Omron CX-Programmer project NewProject (CX-Programmer 9.73)

# PLC NewPLC1: CP1E N20

## Global symbols (name address type ; comment)
0.01 BOOL  ; PB START
100.00 BOOL  ; OUTPUT
100.04 BOOL  ; OUTPUT 2
T001 BOOL  ; TIMER
T002 BOOL  ; TIMER2

## Program NewProgram1 (cyclic task 0)

### Section Section1

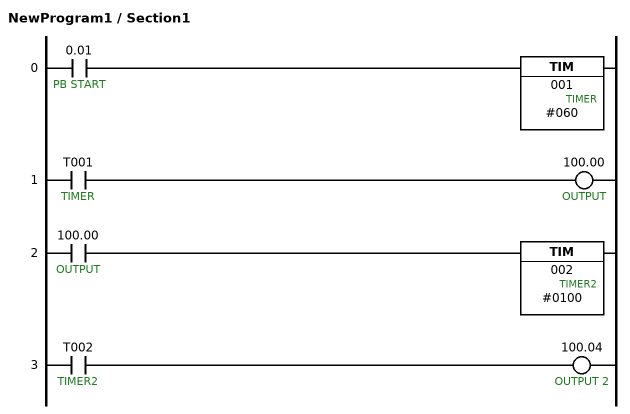
; rung 0
LD 0.01  ; PB START
TIM 001 #060  ; TIMER
; rung 1
LD T001  ; TIMER
OUT 100.00  ; OUTPUT
; rung 2
LD 100.00  ; OUTPUT
TIM 002 #0100  ; TIMER2
; rung 3
LD T002  ; TIMER2
OUT 100.04  ; OUTPUT 2

### Section END
; rung 0
END(001)